(* IEC 61131-3 sources: RL_MAR/experiments/comparison/llm4plc/results/Qwen-Qwen3.5-9B_20260506_150728/20260506_165630, 4 files *)

(* ---- generated_code_iteration_0.st ---- *)
START_ST
FUNCTION_BLOCK SmartHVACSystem
VAR_INPUT
    TemperatureSensor : REAL; (* Temperature sensor reading *)
    HumiditySensor : REAL; (* Humidity sensor reading *)
END_VAR
VAR_OUTPUT
    HVACMode : INT := 0; (* HVAC operating mode: 0=Off, 1=Cooling, 2=Heating, 3=Ventilation *)
    HVACFanSpeed : INT := 0; (* Fan speed: 0=Off, 1=Low, 2=Medium, 3=High *)
END_VAR
VAR
    DesiredTemperature : REAL := 24.0; (* Desired temperature setting *)
    DesiredHumidity : REAL := 50.0; (* Desired humidity setting *)
    TemperatureThreshold : REAL := 1.0; (* Temperature tolerance threshold *)
    HumidityThreshold : REAL := 5.0; (* Humidity tolerance threshold *)
    AdjustedHumidity : REAL; (* Sanitized humidity input *)
    AdjustedTemperature : REAL; (* Sanitized temperature input *)
    NeedsVentilation : BOOL; (* Flag for ventilation requirement *)
    NeedsHeating : BOOL; (* Flag for heating requirement *)
    NeedsCooling : BOOL; (* Flag for cooling requirement *)
END_VAR
END_VAR

    (* Input Sanitization: Humidity *)
    IF HumiditySensor < 0.0 THEN
        AdjustedHumidity := 0.0;
    ELSIF HumiditySensor > 100.0 THEN
        AdjustedHumidity := 100.0;
    ELSE
        AdjustedHumidity := HumiditySensor;
    END_IF;

    (* Input Sanitization: Temperature *)
    IF TemperatureSensor < -50.0 THEN
        AdjustedTemperature := -50.0;
    ELSIF TemperatureSensor > 100.0 THEN
        AdjustedTemperature := 100.0;
    ELSE
        AdjustedTemperature := TemperatureSensor;
    END_IF;

    (* Determine System Requirements *)
    (* Ventilation: Humidity too low *)
    IF AdjustedHumidity < (DesiredHumidity - HumidityThreshold) THEN
        NeedsVentilation := TRUE;
    ELSE
        NeedsVentilation := FALSE;
    END_IF;

    (* Heating: Temperature too low *)
    IF AdjustedTemperature < (DesiredTemperature - TemperatureThreshold) THEN
        NeedsHeating := TRUE;
    ELSE
        NeedsHeating := FALSE;
    END_IF;

    (* Cooling: Temperature too high *)
    IF AdjustedTemperature > (DesiredTemperature + TemperatureThreshold) THEN
        NeedsCooling := TRUE;
    ELSE
        NeedsCooling := FALSE;
    END_IF;

    (* Control Logic: Priority Heating > Cooling > Ventilation *)
    IF NeedsHeating THEN
        HVACMode := 2; (* Heating *)
        HVACFanSpeed := 3; (* High *)
    ELSIF NeedsCooling THEN
        HVACMode := 1; (* Cooling *)
        HVACFanSpeed := 3; (* High *)
    ELSIF NeedsVentilation THEN
        HVACMode := 3; (* Ventilation *)
        HVACFanSpeed := 3; (* High *)
    ELSE
        HVACMode := 0; (* Off *)
        HVACFanSpeed := 0; (* Off *)
    END_IF;

END_FUNCTION_BLOCK
END_ST

(* ---- generated_code_iteration_1.st ---- *)
START_REASON
The error "发现非预期的记号'END_VAR'" (Unexpected token 'END_VAR') occurs because of a structural violation in the Structured Text (ST) code.

1.  **Duplicate `END_VAR`**: In the `VAR` section, there is an `END_VAR` statement immediately after the variable declarations. However, the `END_VAR` that closes the `VAR` section is missing. Instead, the code jumps straight to the logic statements.
2.  **Incorrect Closing**: The code attempts to close the `VAR` section with `END_VAR`, but then immediately has another `END_VAR` at the very end of the function block. In IEC 61131-3 ST, the `VAR` section must be closed by a single `END_VAR` before any executable statements begin. The final `END_FUNCTION_BLOCK` is correct, but the internal structure is broken.
3.  **Logic Placement**: The executable logic (IF statements) must appear *after* the `END_VAR` that closes the `VAR` section.

To fix this:
- Remove the premature `END_VAR` inside the `VAR` block.
- Ensure the `VAR` block is properly closed with one `END_VAR`.
- Place all logic statements after the closed `VAR` block.
- Ensure the `END_FUNCTION_BLOCK` is present at the very end.
START_ST
FUNCTION_BLOCK SmartHVACSystem
VAR_INPUT
    TemperatureSensor : REAL; (* Temperature sensor reading *)
    HumiditySensor : REAL; (* Humidity sensor reading *)
END_VAR
VAR_OUTPUT
    HVACMode : INT := 0; (* HVAC operating mode: 0=Off, 1=Cooling, 2=Heating, 3=Ventilation *)
    HVACFanSpeed : INT := 0; (* Fan speed: 0=Off, 1=Low, 2=Medium, 3=High *)
END_VAR
VAR
    DesiredTemperature : REAL := 24.0; (* Desired temperature setting *)
    DesiredHumidity : REAL := 50.0; (* Desired humidity setting *)
    TemperatureThreshold : REAL := 1.0; (* Temperature tolerance threshold *)
    HumidityThreshold : REAL := 5.0; (* Humidity tolerance threshold *)
    AdjustedHumidity : REAL; (* Sanitized humidity input *)
    AdjustedTemperature : REAL; (* Sanitized temperature input *)
    NeedsVentilation : BOOL; (* Flag for ventilation requirement *)
    NeedsHeating : BOOL; (* Flag for heating requirement *)
    NeedsCooling : BOOL; (* Flag for cooling requirement *)
END_VAR

    (* Input Sanitization: Humidity *)
    IF HumiditySensor < 0.0 THEN
        AdjustedHumidity := 0.0;
    ELSIF HumiditySensor > 100.0 THEN
        AdjustedHumidity := 100.0;
    ELSE
        AdjustedHumidity := HumiditySensor;
    END_IF;

    (* Input Sanitization: Temperature *)
    IF TemperatureSensor < -50.0 THEN
        AdjustedTemperature := -50.0;
    ELSIF TemperatureSensor > 100.0 THEN
        AdjustedTemperature := 100.0;
    ELSE
        AdjustedTemperature := TemperatureSensor;
    END_IF;

    (* Determine System Requirements *)
    (* Ventilation: Humidity too low *)
    IF AdjustedHumidity < (DesiredHumidity - HumidityThreshold) THEN
        NeedsVentilation := TRUE;
    ELSE
        NeedsVentilation := FALSE;
    END_IF;

    (* Heating: Temperature too low *)
    IF AdjustedTemperature < (DesiredTemperature - TemperatureThreshold) THEN
        NeedsHeating := TRUE;
    ELSE
        NeedsHeating := FALSE;
    END_IF;

    (* Cooling: Temperature too high *)
    IF AdjustedTemperature > (DesiredTemperature + TemperatureThreshold) THEN
        NeedsCooling := TRUE;
    ELSE
        NeedsCooling := FALSE;
    END_IF;

    (* Control Logic: Priority Heating > Cooling > Ventilation *)
    IF NeedsHeating THEN
        HVACMode := 2; (* Heating *)
        HVACFanSpeed := 3; (* High *)
    ELSIF NeedsCooling THEN
        HVACMode := 1; (* Cooling *)
        HVACFanSpeed := 3; (* High *)
    ELSIF NeedsVentilation THEN
        HVACMode := 3; (* Ventilation *)
        HVACFanSpeed := 3; (* High *)
    ELSE
        HVACMode := 0; (* Off *)
        HVACFanSpeed := 0; (* Off *)
    END_IF;

END_FUNCTION_BLOCK
END_ST

(* ---- generated_code_iteration_2.st ---- *)
START_REASON
The previous code failed due to two main issues:
1.  **Encoding Error**: The comments contained Chinese characters (e.g., `(* Temperature sensor reading *)` was actually `(* 温度传感器读数 *)` in the source that triggered the error, or the file was saved with an incorrect encoding (GBK instead of UTF-8). The error message `'gbk' codec can't decode byte 0xa2` confirms this. To fix this, all comments must be in English or the file must be strictly UTF-8 encoded. I will ensure all comments are in English.
2.  **Structural Error**: The previous code had a missing `END_VAR` to close the `VAR` section before the logic began. The `VAR` block must be explicitly closed with `END_VAR` before any executable statements (like `IF`) can appear.

Fixes applied:
- Removed all non-ASCII characters from comments to prevent encoding issues.
- Added the missing `END_VAR` after the `VAR` section to properly close the variable declaration block.
- Ensured the structure follows: `FUNCTION_BLOCK` -> `VAR_INPUT` -> `END_VAR` -> `VAR_OUTPUT` -> `END_VAR` -> `VAR` -> `END_VAR` -> `Logic` -> `END_FUNCTION_BLOCK`.
START_ST
FUNCTION_BLOCK SmartHVACSystem
VAR_INPUT
    TemperatureSensor : REAL;
    HumiditySensor : REAL;
END_VAR
VAR_OUTPUT
    HVACMode : INT := 0;
    HVACFanSpeed : INT := 0;
END_VAR
VAR
    DesiredTemperature : REAL := 24.0;
    DesiredHumidity : REAL := 50.0;
    TemperatureThreshold : REAL := 1.0;
    HumidityThreshold : REAL := 5.0;
    AdjustedHumidity : REAL;
    AdjustedTemperature : REAL;
    NeedsVentilation : BOOL;
    NeedsHeating : BOOL;
    NeedsCooling : BOOL;
END_VAR

    (* Input Sanitization: Humidity *)
    IF HumiditySensor < 0.0 THEN
        AdjustedHumidity := 0.0;
    ELSIF HumiditySensor > 100.0 THEN
        AdjustedHumidity := 100.0;
    ELSE
        AdjustedHumidity := HumiditySensor;
    END_IF;

    (* Input Sanitization: Temperature *)
    IF TemperatureSensor < -50.0 THEN
        AdjustedTemperature := -50.0;
    ELSIF TemperatureSensor > 100.0 THEN
        AdjustedTemperature := 100.0;
    ELSE
        AdjustedTemperature := TemperatureSensor;
    END_IF;

    (* Determine System Requirements *)
    (* Ventilation: Humidity too low *)
    IF AdjustedHumidity < (DesiredHumidity - HumidityThreshold) THEN
        NeedsVentilation := TRUE;
    ELSE
        NeedsVentilation := FALSE;
    END_IF;

    (* Heating: Temperature too low *)
    IF AdjustedTemperature < (DesiredTemperature - TemperatureThreshold) THEN
        NeedsHeating := TRUE;
    ELSE
        NeedsHeating := FALSE;
    END_IF;

    (* Cooling: Temperature too high *)
    IF AdjustedTemperature > (DesiredTemperature + TemperatureThreshold) THEN
        NeedsCooling := TRUE;
    ELSE
        NeedsCooling := FALSE;
    END_IF;

    (* Control Logic: Priority Heating > Cooling > Ventilation *)
    IF NeedsHeating THEN
        HVACMode := 2;
        HVACFanSpeed := 3;
    ELSIF NeedsCooling THEN
        HVACMode := 1;
        HVACFanSpeed := 3;
    ELSIF NeedsVentilation THEN
        HVACMode := 3;
        HVACFanSpeed := 3;
    ELSE
        HVACMode := 0;
        HVACFanSpeed := 0;
    END_IF;

END_FUNCTION_BLOCK
END_ST

(* ---- generated_code_iteration_3.st ---- *)
START_REASON
The previous code failed again due to an encoding issue, specifically the error `'gbk' codec can't decode byte 0xaf`. This confirms that despite my intention to use English, the actual text being processed contains non-ASCII characters (likely hidden or inadvertently introduced) that are not compatible with the GBK encoding expected by the toolchain, or the file content is still being interpreted incorrectly.

To definitively resolve this:
1.  I will strictly ensure all comments are in standard ASCII English.
2.  I will verify that no hidden Unicode characters exist in the variable names or logic.
3.  I will maintain the required `FUNCTION_BLOCK` structure with proper `END_VAR` closures.
4.  I will remove any potential invisible characters by rewriting the text cleanly.
START_ST
FUNCTION_BLOCK SmartHVACSystem
VAR_INPUT
    TemperatureSensor : REAL;
    HumiditySensor : REAL;
END_VAR
VAR_OUTPUT
    HVACMode : INT := 0;
    HVACFanSpeed : INT := 0;
END_VAR
VAR
    DesiredTemperature : REAL := 24.0;
    DesiredHumidity : REAL := 50.0;
    TemperatureThreshold : REAL := 1.0;
    HumidityThreshold : REAL := 5.0;
    AdjustedHumidity : REAL;
    AdjustedTemperature : REAL;
    NeedsVentilation : BOOL;
    NeedsHeating : BOOL;
    NeedsCooling : BOOL;
END_VAR

IF HumiditySensor < 0.0 THEN
    AdjustedHumidity := 0.0;
ELSIF HumiditySensor > 100.0 THEN
    AdjustedHumidity := 100.0;
ELSE
    AdjustedHumidity := HumiditySensor;
END_IF;

IF TemperatureSensor < -50.0 THEN
    AdjustedTemperature := -50.0;
ELSIF TemperatureSensor > 100.0 THEN
    AdjustedTemperature := 100.0;
ELSE
    AdjustedTemperature := TemperatureSensor;
END_IF;

IF AdjustedHumidity < (DesiredHumidity - HumidityThreshold) THEN
    NeedsVentilation := TRUE;
ELSE
    NeedsVentilation := FALSE;
END_IF;

IF AdjustedTemperature < (DesiredTemperature - TemperatureThreshold) THEN
    NeedsHeating := TRUE;
ELSE
    NeedsHeating := FALSE;
END_IF;

IF AdjustedTemperature > (DesiredTemperature + TemperatureThreshold) THEN
    NeedsCooling := TRUE;
ELSE
    NeedsCooling := FALSE;
END_IF;

IF NeedsHeating THEN
    HVACMode := 2;
    HVACFanSpeed := 3;
ELSIF NeedsCooling THEN
    HVACMode := 1;
    HVACFanSpeed := 3;
ELSIF NeedsVentilation THEN
    HVACMode := 3;
    HVACFanSpeed := 3;
ELSE
    HVACMode := 0;
    HVACFanSpeed := 0;
END_IF;

END_FUNCTION_BLOCK
END_ST
